// TIA Portal V17 export
// export: Created 2022-07-16T16:56:11.7426569Z, ExportSetting WithDefaults, DisplayName Totally Integrated Automation Portal, DisplayVersion V17, DisplayName TIA Portal Openness, DisplayVersion V17, DisplayName TIA Portal Version Control Interface, DisplayVersion V17, DisplayName TIA Portal Test Suite Advanced, DisplayVersion V17, DisplayName STEP 7 Professional, DisplayVersion V17, DisplayName STEP 7 Safety, DisplayVersion V17, DisplayName WinCC Professional, DisplayVersion V17
TYPE "Client interface_1.Read list"
// stored: IsFailsafeCompliant false
   STRUCT
      SV1scaledValeu { ExternalWritable := 'False'} : Int;
      SV1rawValue { ExternalWritable := 'False'} : Int;
      SV2scaledValeu { ExternalWritable := 'False'} : Int;
      SV2rawValue { ExternalWritable := 'False'} : Int;
      SV3scaledValeu { ExternalWritable := 'False'} : Int;
      SV3rawValue { ExternalWritable := 'False'} : Int;
      value { ExternalWritable := 'False'; S7_SetPoint := 'True'} : "Client interface_1.dbData.value";
      postTestResult { ExternalWritable := 'False'; S7_SetPoint := 'True'} : "Client interface_1.dbData.postTestResult";
      SQactiveSequenceComplete { ExternalWritable := 'False'} : Bool;
      SQactiveSequenceFailed { ExternalWritable := 'False'} : Bool;
      SQpreTestSequenceActive { ExternalWritable := 'False'} : Bool;
      SQmainSequenceActive { ExternalWritable := 'False'} : Bool;
      otherPressure { ExternalWritable := 'False'; S7_SetPoint := 'True'} : "Client interface_1.udtOtherPressure";
   END_STRUCT;
END_TYPE
